FUNCTION_BLOCK FB_StationBase IMPLEMENTS I_Station


VAR
	stMoveOnTrackParameters 	: ST_MoveOnTrackOptions; 
	stMoveRotateOptions	: ST_MoveCOptions; 	
	stStationPosition	: ST_StationPosition;	
	eProcessMode		: E_ProcessMode;
	StationPosition     : PositionXYC;	
	stMoveToPositionOptions: ST_MoveToPositionOptions;
	stJoinTrackOptions: ST_JoinTrackOptions;
	stLeaveTrackOptions: ST_LeaveTrackOptions;
	
	idx  				: UDINT;
	nStateInit			: UDINT;
	nStateClear 		: UDINT;
	nStateProcess		: UDINT;
	bStationInitDone	: BOOL;	
	
	
	// Lists for Stations
	fbList_Station		: FB_List;
	fbList_InputW		: FB_List;		
	fbList_InputS		: FB_List;	
	fbList_InputE		: FB_List;		
	fbList_InputN		: FB_List;	
	
	// History info for debugging purpose
	strInfo				: STRING;	
	fbHistoryInfo		: FB_HistoryInfo;	
	
	
	nProcessRequest		: DINT;
	nProcessClearence	: DINT;
	nProcessState		: UDINT;
	
	fStationPositionOnTrack		: LREAL;	
	
	// =========================
	nStationIndex				: UINT;
	
	nPreviousStationIndexInputW : UINT;	
	nTrackIndexInputW 			: UINT;		
	nPreviousStationIndexInputS : UINT;	
	nTrackIndexInputS 			: UINT;		
	nPreviousStationIndexInputE : UINT;	
	nTrackIndexInputE 			: UINT;		
	nPreviousStationIndexInputN : UINT;	
	nTrackIndexInputN 			: UINT;		
	
	nNextStationIndexOutputW 	: UINT;	
	nTrackIndexOutputW 			: UINT;		
	nNextStationIndexOutputS 	: UINT;	
	nTrackIndexOutputS 			: UINT;		
	nNextStationIndexOutputE 	: UINT;	
	nTrackIndexOutputE 			: UINT;		
	nNextStationIndexOutputN 	: UINT;	
	nTrackIndexOutputN 			: UINT;
	
	fStationPosition_X 			: LREAL;
	fStationPosition_Y 			: LREAL;
	fInRangeDistance			: LREAL;	
	
	fSendAwayDistanceOutputW    : LREAL;	  
    fSendAwayDistanceOutputS    : LREAL;
	fSendAwayDistanceOutputE    : LREAL;	
	fSendAwayDistanceOutputN    : LREAL;
	
	fSendAwayPositionOutputW	: LREAL;
	fSendAwayPositionOutputS	: LREAL;
	fSendAwayPositionOutputE	: LREAL;
	fSendAwayPositionOutputN	: LREAL;	
	
	nStationTrackIndex			: UINT;
	nStationTaskList              :ARRAY[1..200] OF  UDINT;

	position					: PositionXYC;

	// communication data
	bComEnable			: BOOL;
	bComProcessComplete: BOOL;
	bComOK				: BOOL;
	bComNOK				: BOOL;
	bComError			: BOOL;
	nComStatusWord		: INT;
	nComErrorID			: INT;
	sComProcesedMover	: STRING(13);
	aComMoversList		: ARRAY[1..10] OF STRING(13);
	nComControlWord		: INT;
END_VAR

METHOD Clear : BOOL
VAR_INPUT
END_VAR


VAR_INST

	nStateClear : UINT;

END_VAR


	CASE nStateClear OF 
		
	0:	// Enter
		            Clear := FALSE;
		  nProcessRequest := 0;
		nProcessClearence := 0;
		    nProcessState := 0;	  
			  
		nStateClear := nStateClear +10;
		
	10: // Clear Station-List
		IF fbList_Station.ClearList() THEN
			nStateClear := nStateClear +10;	
		END_IF
		
	20: // Clear InputW-List
		IF fbList_InputW.ClearList() THEN
			nStateClear := nStateClear +10;	
		END_IF
	
	30: // Clear InputE-List
		IF fbList_InputE.ClearList() THEN
			nStateClear := nStateClear +10;	
		END_IF	
	
	40: // Clear InputS-List
		IF fbList_InputS.ClearList() THEN
			nStateClear := nStateClear +10;	
		END_IF		
	
	50: // Clear InputN-List
		IF fbList_InputN.ClearList() THEN
			nStateClear := nStateClear +10;	
		END_IF
	
	60:	nStateClear := 100;	
		
		
	100:  // Done
		nStateClear := 0;
		      Clear := TRUE;
		
	END_CASE
END_METHOD

METHOD Cycle : BOOL
VAR_INPUT
END_VAR
VAR
	nForCounter : INT;
END_VAR


VAR_INST
	
	fTestValueX	: LREAL;
	fTestValueY : LREAL;	
	
END_VAR
IF communication.RunAplicationComm AND nStationIndex > 0 AND nStationIndex <= GVL.gc_NumberStations THEN

    Communication.g_Com_Stations[nStationIndex].OUT.Enable := bComEnable;
    Communication.g_Com_Stations[nStationIndex].OUT.ProcessComplete := bComProcessComplete;
    Communication.g_Com_Stations[nStationIndex].OUT.OK := bComOK;
    Communication.g_Com_Stations[nStationIndex].OUT.NOK := bComNOK;
    Communication.g_Com_Stations[nStationIndex].OUT.Error := bComError;
    Communication.g_Com_Stations[nStationIndex].OUT.StatusWord := nComStatusWord;
    Communication.g_Com_Stations[nStationIndex].OUT.StationName := nStationIndex;
    Communication.g_Com_Stations[nStationIndex].OUT.Error_ID := nComErrorID;
    Communication.g_Com_Stations[nStationIndex].OUT.ProcesedMover := sComProcesedMover;
    Communication.g_Com_Stations[nStationIndex].OUT.MoversList := aComMoversList;

    nComControlWord := Communication.g_Com_Stations[nStationIndex].IN.ControlWord;

END_IF
END_METHOD

METHOD Init : BOOL


	  nStateInit := 0;
	nStateProcess := 0;
	 eProcessMode := E_ProcessMode.None;

	Init := TRUE;
END_METHOD

PROPERTY P_bInitDone : BOOL
GET
P_bInitDone := bStationInitDone;
END_GET
END_PROPERTY

PROPERTY P_eProcessMode : E_ProcessMode
GET
P_eProcessMode := eProcessMode;
END_GET
SET
eProcessMode := P_eProcessMode;
END_SET
END_PROPERTY

PROPERTY P_List_Station : I_List
GET
P_List_Station := fbList_Station;
END_GET
END_PROPERTY

PROPERTY P_List_Switch_Input_E : I_List
GET
P_List_Switch_Input_E := fbList_InputE;
END_GET
END_PROPERTY

{warning 'Add property implementation'}
PROPERTY P_List_Switch_Input_N : I_List
GET
P_List_Switch_Input_N := fbList_InputN;
END_GET
END_PROPERTY

PROPERTY P_List_Switch_Input_S : I_List
GET
P_List_Switch_Input_S := fbList_InputS;
END_GET
END_PROPERTY

PROPERTY P_List_Switch_Input_W : I_List
GET
P_List_Switch_Input_W := fbList_InputW;
END_GET
END_PROPERTY

PROPERTY P_nErrorCode : UDINT
GET
END_GET
END_PROPERTY

PROPERTY P_Position : ST_StationPosition
GET
P_Position := stStationPosition;
END_GET
END_PROPERTY

PROPERTY P_ProcessClearance : DINT
GET
P_ProcessClearance := nProcessClearence;
END_GET
END_PROPERTY

PROPERTY P_ProcessRequest : UDINT
GET
P_ProcessRequest := nProcessRequest;
END_GET
SET
nProcessRequest := P_ProcessRequest;
END_SET
END_PROPERTY

PROPERTY P_ProcessState : UDINT
GET
P_ProcessState := nProcessState;
END_GET
SET
nProcessState := P_ProcessState;
END_SET
END_PROPERTY

PROPERTY P_StationTaskList : array[1..200] of UDINT
GET
 P_StationTaskList := nStationTaskList;
END_GET
SET
nStationTaskList := P_StationTaskList;
END_SET
END_PROPERTY

PROPERTY P_Enable : BOOL
GET
P_Enable := bComEnable;
END_GET
SET
bComEnable := P_Enable;
END_SET
END_PROPERTY

PROPERTY P_ProcessComplete : BOOL
GET
P_ProcessComplete := bComProcessComplete;
END_GET
SET
bComProcessComplete := P_ProcessComplete;
END_SET
END_PROPERTY

PROPERTY P_OK : BOOL
GET
P_OK := bComOK;
END_GET
SET
bComOK := P_OK;
END_SET
END_PROPERTY

PROPERTY P_NOK : BOOL
GET
P_NOK := bComNOK;
END_GET
SET
bComNOK := P_NOK;
END_SET
END_PROPERTY

PROPERTY P_ComError : BOOL
GET
P_ComError := bComError;
END_GET
SET
bComError := P_ComError;
END_SET
END_PROPERTY

PROPERTY P_StatusWord : INT
GET
P_StatusWord := nComStatusWord;
END_GET
SET
nComStatusWord := P_StatusWord;
END_SET
END_PROPERTY

PROPERTY P_ComErrorID : INT
GET
P_ComErrorID := nComErrorID;
END_GET
SET
nComErrorID := P_ComErrorID;
END_SET
END_PROPERTY

PROPERTY P_ProcesedMover : STRING(13)
GET
P_ProcesedMover := sComProcesedMover;
END_GET
SET
sComProcesedMover := P_ProcesedMover;
END_SET
END_PROPERTY

PROPERTY P_MoversList : ARRAY[1..10] OF STRING(13)
GET
P_MoversList := aComMoversList;
END_GET
SET
aComMoversList := P_MoversList;
END_SET
END_PROPERTY

PROPERTY P_ControlWord : INT
GET
P_ControlWord := nComControlWord;
END_GET
SET
nComControlWord := P_ControlWord;
END_SET
END_PROPERTY

METHOD Process : BOOL
END_METHOD

END_FUNCTION_BLOCK

(* stored: Version 1.1.0.1
   POU FB_StationBase: Id {2d0c860d-5211-414b-ba0b-04cb8f828be8}, SpecialFunc None
   Folder Properties: Id {fd0777f5-fc91-4b83-836b-3df138db01e0}
   Method Clear: Id {4c408367-064c-402d-970b-be8f83eec97f}
   Method Cycle: Id {797df6f0-b770-4dee-8c02-4a52ac49eae5}
   Method Init: Id {85cd9382-c88a-4b80-9e3d-de78cce941af}
   Property P_bInitDone: Id {170fcc51-70b8-40e7-8501-42641c79dd41}
   Get Get: Id {d9b8fa73-a40a-4e02-a707-987591016094}
   Property P_eProcessMode: Id {a54e278b-d4a2-4042-b6f6-2faa9d3150a4}
   Get Get: Id {2d664a2f-5618-4f32-864a-2b78419db8d4}
   Set Set: Id {da929ff5-0a0a-43f0-b0fd-4a7332f4a163}
   Property P_List_Station: Id {3671176d-73b2-4e4e-b189-17340f7a85ec}
   Get Get: Id {35e420ae-5ee2-43c4-8018-524c39f926db}
   Property P_List_Switch_Input_E: Id {82605b03-ce95-4909-86ba-594ecd6e3795}
   Get Get: Id {4841efdc-0d89-457a-ba5a-c71197c1a8f2}
   Property P_List_Switch_Input_N: Id {499ed030-b0e7-4dd9-88fd-d75590656591}
   Get Get: Id {9e04b48f-2188-4c67-85b2-402b3e4920c2}
   Property P_List_Switch_Input_S: Id {ce1be437-a7e0-466f-95d5-40b68723035a}
   Get Get: Id {fe5495c0-2c20-49e5-87b6-79da5cfd19da}
   Property P_List_Switch_Input_W: Id {41e14359-4087-4409-aa1f-5e851e1896f0}
   Get Get: Id {f84852de-8fb1-48db-bf90-81dca3b69d94}
   Property P_nErrorCode: Id {4695a954-7f43-4461-9ea0-ed2a17d7feef}
   Get Get: Id {3bfef907-5a1d-4fbc-8e70-173f2d934fdb}
   Property P_Position: Id {6fa15b1b-62e2-4bcd-948c-68774bb7cd41}
   Get Get: Id {e4f1bd5d-1a08-4b5b-946c-d545bafad611}
   Property P_ProcessClearance: Id {89046516-3382-4aba-9276-635fdf14ed66}
   Get Get: Id {2a88829c-57bb-44c8-a204-1ae062ca71c0}
   Property P_ProcessRequest: Id {6ac380ee-8832-4c4c-97a8-197f9b499c3b}
   Get Get: Id {df7ccd5e-4155-464a-a8a5-2efbf0b8422f}
   Set Set: Id {02fa14bf-51b1-4bb5-b432-e7b9dc57f354}
   Property P_ProcessState: Id {bc88e717-95c4-49d8-8348-42122813a034}
   Get Get: Id {5b1a7d6f-291b-4705-83c7-530bb8e1d4f9}
   Set Set: Id {bc1e3dd3-dac7-42d8-99c3-e55c1cafdb1d}
   Property P_StationTaskList: Id {e2530656-5473-4313-8444-ebeb2bb306db}
   Get Get: Id {11a0ae5e-75b6-4460-bfc7-b0a295ba884c}
   Set Set: Id {f8c6877e-bcc7-4e3a-ad37-ce80d731078b}
   Property P_Enable: Id {c1a2b3d4-1111-4a2b-8c3d-4e5f6a7b8c01}
   Get Get: Id {c1a2b3d4-1111-4a2b-8c3d-4e5f6a7b8c02}
   Set Set: Id {c1a2b3d4-1111-4a2b-8c3d-4e5f6a7b8c03}
   Property P_ProcessComplete: Id {c1a2b3d4-2222-4a2b-8c3d-4e5f6a7b8c01}
   Get Get: Id {c1a2b3d4-2222-4a2b-8c3d-4e5f6a7b8c02}
   Set Set: Id {c1a2b3d4-2222-4a2b-8c3d-4e5f6a7b8c03}
   Property P_OK: Id {c1a2b3d4-3333-4a2b-8c3d-4e5f6a7b8c01}
   Get Get: Id {c1a2b3d4-3333-4a2b-8c3d-4e5f6a7b8c02}
   Set Set: Id {c1a2b3d4-3333-4a2b-8c3d-4e5f6a7b8c03}
   Property P_NOK: Id {c1a2b3d4-4444-4a2b-8c3d-4e5f6a7b8c01}
   Get Get: Id {c1a2b3d4-4444-4a2b-8c3d-4e5f6a7b8c02}
   Set Set: Id {c1a2b3d4-4444-4a2b-8c3d-4e5f6a7b8c03}
   Property P_ComError: Id {c1a2b3d4-5555-4a2b-8c3d-4e5f6a7b8c01}
   Get Get: Id {c1a2b3d4-5555-4a2b-8c3d-4e5f6a7b8c02}
   Set Set: Id {c1a2b3d4-5555-4a2b-8c3d-4e5f6a7b8c03}
   Property P_StatusWord: Id {c1a2b3d4-6666-4a2b-8c3d-4e5f6a7b8c01}
   Get Get: Id {c1a2b3d4-6666-4a2b-8c3d-4e5f6a7b8c02}
   Set Set: Id {c1a2b3d4-6666-4a2b-8c3d-4e5f6a7b8c03}
   Property P_ComErrorID: Id {c1a2b3d4-7777-4a2b-8c3d-4e5f6a7b8c01}
   Get Get: Id {c1a2b3d4-7777-4a2b-8c3d-4e5f6a7b8c02}
   Set Set: Id {c1a2b3d4-7777-4a2b-8c3d-4e5f6a7b8c03}
   Property P_ProcesedMover: Id {c1a2b3d4-8888-4a2b-8c3d-4e5f6a7b8c01}
   Get Get: Id {c1a2b3d4-8888-4a2b-8c3d-4e5f6a7b8c02}
   Set Set: Id {c1a2b3d4-8888-4a2b-8c3d-4e5f6a7b8c03}
   Property P_MoversList: Id {c1a2b3d4-9999-4a2b-8c3d-4e5f6a7b8c01}
   Get Get: Id {c1a2b3d4-9999-4a2b-8c3d-4e5f6a7b8c02}
   Set Set: Id {c1a2b3d4-9999-4a2b-8c3d-4e5f6a7b8c03}
   Property P_ControlWord: Id {c1a2b3d4-aaaa-4a2b-8c3d-4e5f6a7b8c01}
   Get Get: Id {c1a2b3d4-aaaa-4a2b-8c3d-4e5f6a7b8c02}
   Set Set: Id {c1a2b3d4-aaaa-4a2b-8c3d-4e5f6a7b8c03}
   Method Process: Id {aa10b277-24cb-4f44-9514-ef81c196a6e7} *)
